SYSTEM FLASHER_TESTD (* Distributed Flasher Test System Configuration *)
  (* Standard: 61499-1 *)
  (* Version 0.0, 2001-07-31, JHC, Rockwell Automation, Changed IN_TIME to IN_ANY, adjusted height. *)
  (* Version 0.0, 2001-02-22, JHC, Rockwell Automation *)
  APPLICATION TEST
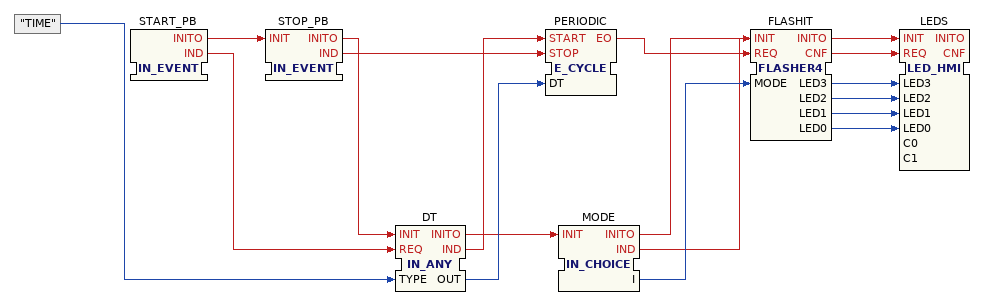
    FBS
      START_PB : IN_EVENT;
      STOP_PB : IN_EVENT;
      DT : IN_ANY;
      PERIODIC : E_CYCLE;
      MODE : IN_CHOICE;
      FLASHIT : FLASHER4;
      LEDS : LED_HMI;
    END_FBS
    EVENT_CONNECTIONS
      START_PB.INITO TO STOP_PB.INIT;
      STOP_PB.INITO TO DT.INIT;
      DT.INITO TO MODE.INIT;
      MODE.INITO TO FLASHIT.INIT;
      FLASHIT.INITO TO LEDS.INIT;
      START_PB.IND TO DT.REQ;
      DT.IND TO PERIODIC.START;
      STOP_PB.IND TO PERIODIC.STOP;
      MODE.IND TO FLASHIT.INIT;
      PERIODIC.EO TO FLASHIT.REQ;
      FLASHIT.CNF TO LEDS.REQ;
    END_CONNECTIONS
    DATA_CONNECTIONS
      DT.OUT TO PERIODIC.DT;
      MODE.I TO FLASHIT.MODE;
      FLASHIT.LED3 TO LEDS.LED3;
      FLASHIT.LED2 TO LEDS.LED2;
      FLASHIT.LED1 TO LEDS.LED1;
      FLASHIT.LED0 TO LEDS.LED0;
      "TIME" TO DT.TYPE;
    END_CONNECTIONS
  END_APPLICATION
  DEVICE FLASHER : FRAME_DEVICE
    RESOURCE RES1 : PANEL_RESOURCE
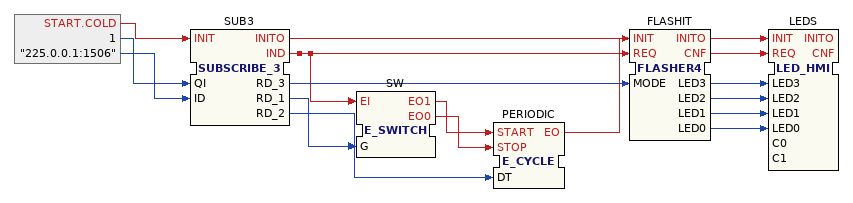
      FBS
        SUB3 : SUBSCRIBE_3;
        SW : E_SWITCH;
        PERIODIC : E_CYCLE;
        FLASHIT : FLASHER4;
        LEDS : LED_HMI;
      END_FBS
      EVENT_CONNECTIONS
        START.COLD TO SUB3.INIT;
        SUB3.INITO TO FLASHIT.INIT;
        FLASHIT.INITO TO LEDS.INIT;
        SUB3.IND TO SW.EI;
        SW.EO1 TO PERIODIC.START;
        SW.EO0 TO PERIODIC.STOP;
        SUB3.IND TO FLASHIT.INIT;
        PERIODIC.EO TO FLASHIT.REQ;
        FLASHIT.CNF TO LEDS.REQ;
      END_CONNECTIONS
      DATA_CONNECTIONS
        SUB3.RD_3 TO FLASHIT.MODE;
        FLASHIT.LED3 TO LEDS.LED3;
        FLASHIT.LED2 TO LEDS.LED2;
        FLASHIT.LED1 TO LEDS.LED1;
        FLASHIT.LED0 TO LEDS.LED0;
        1 TO SUB3.QI;
        SUB3.RD_1 TO SW.G;
        SUB3.RD_2 TO PERIODIC.DT;
        "225.0.0.1:1506" TO SUB3.ID;
      END_CONNECTIONS
    END_RESOURCE
    DATA_CONNECTIONS
      0 TO RES1.TRACE;
    END_CONNECTIONS
  END_DEVICE
  DEVICE CTL_PANEL : FRAME_DEVICE
    RESOURCE RES1 : PANEL_RESOURCE
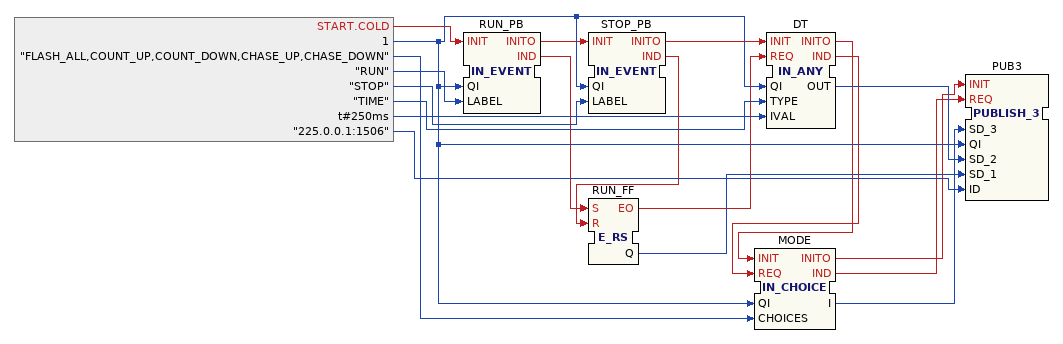
      FBS
        RUN_PB : IN_EVENT;
        STOP_PB : IN_EVENT;
        RUN_FF : E_RS;
        MODE : IN_CHOICE;
        DT : IN_ANY;
        PUB3 : PUBLISH_3;
      END_FBS
      EVENT_CONNECTIONS
        START.COLD TO RUN_PB.INIT;
        RUN_PB.INITO TO STOP_PB.INIT;
        STOP_PB.INITO TO DT.INIT;
        DT.INITO TO MODE.INIT;
        MODE.INITO TO PUB3.INIT;
        RUN_PB.IND TO RUN_FF.S;
        STOP_PB.IND TO RUN_FF.R;
        RUN_FF.EO TO DT.REQ;
        DT.IND TO MODE.REQ;
        MODE.IND TO PUB3.REQ;
      END_CONNECTIONS
      DATA_CONNECTIONS
        1 TO MODE.QI;
        MODE.I TO PUB3.SD_3;
        "FLASH_ALL,COUNT_UP,COUNT_DOWN,CHASE_UP,CHASE_DOWN" TO MODE.CHOICES;
        1 TO RUN_PB.QI;
        "RUN" TO RUN_PB.LABEL;
        1 TO DT.QI;
        1 TO STOP_PB.QI;
        "STOP" TO STOP_PB.LABEL;
        1 TO PUB3.QI;
        DT.OUT TO PUB3.SD_2;
        RUN_FF.Q TO PUB3.SD_1;
        "TIME" TO DT.TYPE;
        t#250ms TO DT.IVAL;
        "225.0.0.1:1506" TO PUB3.ID;
      END_CONNECTIONS
    END_RESOURCE
    DATA_CONNECTIONS
      0 TO RES1.TRACE;
    END_CONNECTIONS
  END_DEVICE
  DATA_CONNECTIONS (* parameter values *)
    [1,1] TO FLASHER.GRID;
    [280,100,225,75] TO FLASHER.BOUNDS;
    [50,100,225,100] TO CTL_PANEL.BOUNDS;
    [1,1] TO CTL_PANEL.GRID;
  END_CONNECTIONS
END_SYSTEM
